FUNCTION_BLOCK TcoDatamanRead_v_5_x_x EXTENDS TcoCore.TcoTask
VAR_IN_OUT
    inoIoData : TcoDatamanIO_v_5_x_x;
    inoConfig : TcoDatamanConfig_v_5_x_x;
    inoStatus : TcoDatamanStatus_v_5_x_x;
    inoResults : TcoDatamanResults_v_5_x_x;
END_VAR
VAR
    {attribute 'hide'}
    _progress : INT := 0;
    {attribute 'hide'}
    _infoTimer : TON;
    {attribute 'hide'}
    _errorTimer : TON;
    {attribute 'hide'}
    _varInfo : __SYSTEM.VAR_INFO;
    {attribute 'hide'}
    _sb : TcoCore.StringBuilder;
END_VAR

IF Execute() THEN
    IF _progress = 0 THEN
        IF NOT __ISVALIDREF(inoIoData) THEN
            _varInfo := __VARINFO(inoIoData);
            Messenger.Programming(_sb.Clear().Append('<#Invalid reference: #>').Append(_varInfo.Symbol).ToString()).Pin();
        ELSIF NOT __ISVALIDREF(inoConfig) THEN
            _varInfo := __VARINFO(inoConfig);
            Messenger.Programming(_sb.Clear().Append('<#Invalid reference: #>').Append(_varInfo.Symbol).ToString()).Pin();
        ELSIF NOT __ISVALIDREF(inoStatus) THEN
            _varInfo := __VARINFO(inoStatus);
            Messenger.Programming(_sb.Clear().Append('<#Invalid reference: #>').Append(_varInfo.Symbol).ToString()).Pin();
        ELSIF NOT __ISVALIDREF(inoResults) THEN
            _varInfo := __VARINFO(inoResults);
            Messenger.Programming(_sb.Clear().Append('<#Invalid reference: #>').Append(_varInfo.Symbol).ToString()).Pin();
        ELSE
            _progress := _progress + 1;
        END_IF
    END_IF

    IF _progress = 1 THEN
        THIS^.inoStatus.ActionDescription := '<#Reading running.#>';
        CallTimers(FALSE);
        _progress := _progress + 1;
    END_IF

    IF _progress = 2 THEN
        THIS^.inoIoData.AcquisitionControl.TriggerEnable := TRUE;
        THIS^.inoIoData.AcquisitionControl.Trigger := FALSE;
        THIS^.inoIoData.ResultsControl.EnableResultBuffering := FALSE;
        THIS^.inoIoData.ResultsControl.ResultsAcknowledge := THIS^.inoIoData.ResultsStatus.ResultsAvailable;
        THIS^.Messenger.OnCondition(_infoTimer.Q).Warning('<#Waiting for the signal ResultsAvailable to be reseted!#>').Pin();

        IF NOT THIS^.inoIoData.ResultsStatus.ResultsAvailable THEN
            CallTimers(FALSE);
            _progress := _progress + 1;
        END_IF
    END_IF

    IF _progress = 3 THEN
        THIS^.Messenger.OnCondition(_infoTimer.Q).Warning('<#Waiting for the signal TriggerReady to be set!#>').Pin();

        IF THIS^.inoIoData.AcquisitionStatus.TriggerReady THEN
            CallTimers(FALSE);
            _progress := _progress + 1;
        END_IF
    END_IF

    IF _progress = 4 THEN
        THIS^.inoIoData.AcquisitionControl.Trigger := TRUE;
        THIS^.Messenger.OnCondition(_infoTimer.Q).Warning('<#Waiting for the signal TriggerAcknowledge to be set!#>').Pin();

        IF THIS^.inoIoData.AcquisitionStatus.TriggerAcknowledge THEN
            CallTimers(FALSE);
            _progress := _progress + 1;
        END_IF
    END_IF

    IF _progress = 5 THEN
        THIS^.Messenger.OnCondition(_infoTimer.Q).Warning('<#Waiting for the signal ResultsAvailable to be set!#>').Pin();

        IF THIS^.inoIoData.ResultsStatus.ResultsAvailable THEN
            CallTimers(FALSE);
            _progress := _progress + 1;
        END_IF
    END_IF

    IF _progress = 6 THEN
        THIS^.inoResults.Length := THIS^.inoIoData.ResultData.ResultLength;
        THIS^.Messenger.OnCondition(_infoTimer.Q).Warning('<#Waiting for the ResultData copied!#>').Pin();

        IF Tc2_System
            .MEMCPY(srcAddr := ADR(THIS^.inoIoData.ResultData.ResultData), destAddr := ADR(THIS^.inoResults.Data), n := THIS^.inoResults.Length) >
            0 AND
            Tc2_System.MEMSET(destAddr :=
                ADR(THIS^.inoResults.Data) + THIS^.inoResults.Length,
                fillByte := 0,
                n := SIZEOF(THIS^.inoResults.Data) - THIS^.inoResults.Length) >
            0 THEN
            CallTimers(FALSE);
            _progress := _progress + 1;
        END_IF
    END_IF

    IF _progress = 7 THEN
        THIS^.inoIoData.AcquisitionControl.Trigger := FALSE;
        THIS^.inoIoData.ResultsControl.EnableResultBuffering := FALSE;
        THIS^.inoIoData.ResultsControl.ResultsAcknowledge := TRUE;
        THIS^.ThrowWhen(THIS^.inoIoData.ResultData.ResultCode = 0 OR THIS^.inoIoData.ResultData.ResultLength = 0);
        THIS^.DoneWhen(TRUE);
        _progress := 0;
    END_IF

    CallTimers(TRUE);
    THIS^.ThrowWhen(_errorTimer.Q);
END_IF

METHOD CallTimers
VAR_INPUT
    inValue : BOOL;
END_VAR
_infoTimer(IN := inValue, PT := THIS^.inoConfig.InfoTime);
_errorTimer(IN := inValue, PT := THIS^.inoConfig.ErrorTime);
END_METHOD

{attribute 'hide'}
METHOD PUBLIC FB_init : BOOL
VAR_INPUT
    bInitRetains : BOOL; // if TRUE, the retain variables are initialized (warm start / cold start)
    bInCopyCode : BOOL; // if TRUE, the instance afterwards gets moved into the copy code (online change)
    ParentObject : ITcoObject;
END_VAR
END_METHOD

(*~
    <docu>
        <summary>
            Executes when task is aborted.
        </summary>
    </docu>
~*)
METHOD PROTECTED OnAbort
THIS^.inoStatus.ActionDescription := '<#Reading was aborted, while not yet completed!#>';
END_METHOD

(*~
    <docu>
        <summary>
            Executes when task reaches the ```Done``` state .
        </summary>
    </docu>
~*)
METHOD PROTECTED OnDone
THIS^.inoStatus.ActionDescription := '<#Reading was completed successfully.#>';
END_METHOD

(*~
    <docu>
        <summary>
            Executes when task reaches the ```Error``` state.
            <para>
                Do not confuse with <see cref="PlcDocu.TcoCore.TcoTask.WhileError()"/>, that is called cyclically until '''Error''' state is left.
            </para>
        </summary>
    </docu>
~*)
METHOD PROTECTED OnError
THIS^.inoStatus.ActionDescription := '<#Reading finished with error.#>';
END_METHOD

METHOD PROTECTED OnStart
THIS^.inoStatus.ActionDescription := '<#Reading started.#>';
THIS^.inoStatus.ResultString := '';
END_METHOD

(*~
    <docu>
        <summary>
            Restores this instance to the Ready state. Can be called explicitly or from within one of the restore mechanisms.
            <para>
                See also <see cref="PlcDocu.TcoCore.TcoTask.AutoRestorable()"/>
            </para>
        </summary>
    </docu>
~*)
METHOD Restore : ITcoRestorable
SUPER^.Restore();
_progress := 0;
CallTimers(FALSE);
Messenger.UnPin();
END_METHOD

END_FUNCTION_BLOCK

(* stored: Version 1.1.0.1, ProductVersion 3.1.4024.12
   POU TcoDatamanRead_v_5_x_x: Id {bbfbdcf8-58e6-0eb9-1267-89fca8b94731}, SpecialFunc None
   Method CallTimers: Id {fe44bf2a-41b1-0036-2ff7-3c71ca913b03}
   Method FB_init: Id {332a4519-fd52-0dcc-3b76-6a8434ca4896}
   Method OnAbort: Id {dc1bb021-ea15-063c-2539-0b643900f778}
   Method OnDone: Id {967e6af2-8a80-0fd1-032f-4a8fa1f0de90}
   Method OnError: Id {c9648a71-225a-0f5c-2a0c-96ef9d7e736f}
   Method OnStart: Id {4897565b-7f96-0e88-026b-65aa04f41ba7}
   Method Restore: Id {84a80bc1-f9a1-02f8-039f-6c297c2533d7} *)
